{region '#Template'}
	{attribute 'Version' := '0.0.1.0'}
	{attribute 'Tags' := '"LCID": "1031", "Text": "DUT, System, UPS"'}
	{attribute 'Tags' := '"LCID": "1033", "Text": "DUT, System, UPS"'}
	{attribute 'Description' := '"LCID": "1031", "Text": "Einstellung USV"'}
	{attribute 'Description' := '"LCID": "1033", "Text": "Settings UPS"'}
{endregion}

{attribute 'qualified_only'}
{attribute 'strict'}
TYPE E_BA_UPSType :
(
	eNone := 0,
	
	eCX50x0,
	eCX51x0,
	eCX81xx,
	eCX9020_U900,
	eCB3011
);
END_TYPE

(* stored: Version 1.1.0.1, ProductVersion 3.1.4024.6
   DUT E_BA_UPSType: Id {10646073-d56c-4e97-a433-6f1c2ad3830a} *)
